SUBAPPLICATION mapping_Uebung_034 (* Analog-Eingang auf PWM Ausgang *)
  (* Standard: 61499-2 *)
  (* Version 1.0, 2023-10-23, franz *)
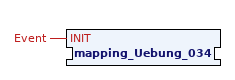
  EVENT_INPUT
    INIT;
  END_EVENT
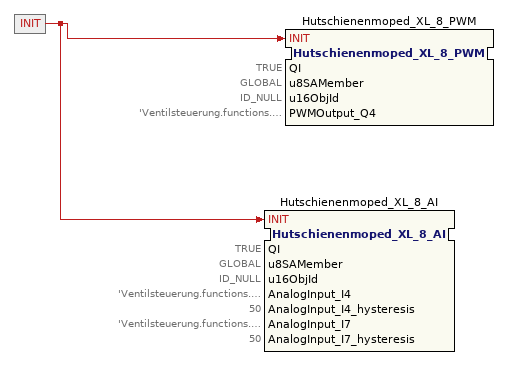
  FBS
    Hutschienenmoped_XL_8_AI : Hutschienenmoped_XL_8_AI(QI := TRUE, u8SAMember := GLOBAL, u16ObjId := ID_NULL, AnalogInput_I4 := 'Ventilsteuerung.functions.AnalogInput_I4', AnalogInput_I4_hysteresis := 50, AnalogInput_I7 := 'Ventilsteuerung.functions.AnalogInput_I7', AnalogInput_I7_hysteresis := 50);
    Hutschienenmoped_XL_8_PWM : Hutschienenmoped_XL_8_PWM(QI := TRUE, u8SAMember := GLOBAL, u16ObjId := ID_NULL, PWMOutput_Q4 := 'Ventilsteuerung.functions.PWMOutput_Q4');
  END_FBS
  EVENT_CONNECTIONS
    INIT TO Hutschienenmoped_XL_8_AI.INIT;
    INIT TO Hutschienenmoped_XL_8_PWM.INIT;
  END_CONNECTIONS
END_SUBAPPLICATION
